{attribute 'GeneratedUsingTerminal: EL5101-0011-0016'}
{attribute addProperty BoxType "EL5101-0011-0016"}
{attribute addProperty Id "Set_counter_doneBOOL1Open_circuitBOOL1Status_of_input_ABOOL1Status_of_input_BBOOL1Status_of_input_CBOOL1Sync_errorBOOL1TxPDO_StateBOOL1TxPDO_ToggleBOOL1"}
{attribute addProperty CRC "775505615"}
{attribute addProperty Size "8"}
TYPE Status_2E3946CF :
STRUCT
	{attribute addProperty Name "Set_counter_done"}
	Set_counter_done : BOOL;
	{attribute addProperty Name "Open_circuit"}
	Open_circuit : BOOL;
	{attribute addProperty Name "Status_of_input_A"}
	Status_of_input_A : BOOL;
	{attribute addProperty Name "Status_of_input_B"}
	Status_of_input_B : BOOL;
	{attribute addProperty Name "Status_of_input_C"}
	Status_of_input_C : BOOL;
	{attribute addProperty Name "Sync_error"}
	Sync_error : BOOL;
	{attribute addProperty Name "TxPDO_State"}
	TxPDO_State : BOOL;
	{attribute addProperty Name "TxPDO_Toggle"}
	TxPDO_Toggle : BOOL;
END_STRUCT
END_TYPE

(* stored: Version 1.2.0.0, ProductVersion 3.1.4024.9
   DUT Status_2E3946CF: Id {08b1b8b0-7c1a-4f96-9d61-f0e66de592c4} *)
